{attribute 'linkalways'} 
{attribute 'no_explicit_call' := 'This FB is a CLASS and must be accessed using methods or properties'}
{attribute 'enable_dynamic_creation'}
FUNCTION_BLOCK _WORD EXTENDS NumericDatatypeBase
VAR
	localData : WORD;
	activeData : REFERENCE TO WORD REF= localData;
END_VAR

PROPERTY PUBLIC Address : PVOID
GET
Address := ADR(activeData);
END_GET
END_PROPERTY

METHOD PUBLIC ClearReference
VAR_INPUT
END_VAR
activeData REF= localData;
END_METHOD

METHOD PUBLIC Clone : I_Datatype
VAR
    pClone : POINTER TO _WORD;
END_VAR
pClone := __NEW(_WORD(InitialValue := Value));
Clone := pClone^;
END_METHOD

METHOD FB_init : BOOL
VAR_INPUT
	bInitRetains : BOOL; // if TRUE, the retain variables are initialized (warm start / cold start)
	bInCopyCode : BOOL;  // if TRUE, the instance afterwards gets moved WORDo the copy code (online change)
	InitialValue : WORD;
END_VAR
localData := InitialValue;
END_METHOD

PROPERTY PUBLIC IsEven : BOOL
GET
IsEven := (Value mod 2) = 0;
END_GET
END_PROPERTY

PROPERTY PUBLIC IsFloat : BOOL
GET
IsFloat := FALSE;
END_GET
END_PROPERTY

PROPERTY PUBLIC IsSigned : BOOL
GET
IsSigned := FALSE;
END_GET
END_PROPERTY

METHOD PUBLIC MakeReferenceTo
VAR_INPUT
	ReferenceTarget : REFERENCE TO WORD;
END_VAR
activeData REF= ReferenceTarget;
END_METHOD

PROPERTY PUBLIC MaxValue : WORD
GET
MaxValue :=  DatatypeLimits.WORD_MAX_VALUE;
END_GET
END_PROPERTY

PROPERTY PUBLIC MinValue : WORD
GET
MinValue := DatatypeLimits.WORD_MIN_VALUE;
END_GET
END_PROPERTY

METHOD PROTECTED SerializeMaxValue
VAR_INPUT
	Serializer : I_Serializer;
END_VAR
Serializer.AddWord(MaxValue);
END_METHOD

METHOD PROTECTED SerializeMinValue
VAR_INPUT
	Serializer : I_Serializer;
END_VAR
Serializer.AddWord(MinValue);
END_METHOD

METHOD PUBLIC SerializeWith
VAR_INPUT
	Serializer : I_Serializer;
END_VAR
Serializer.AddWord(activeData);
END_METHOD

PROPERTY PUBLIC Size : UDINT
GET
Size := SIZEOF(activeData);
END_GET
END_PROPERTY

METHOD TryDeserializeFrom : BOOL
VAR_INPUT
	Deserializer : I_Deserializer;
	Feedback : I_DeserializerFeedback;
END_VAR
TryDeserializeFrom := Deserializer.TryGetWord(activeData, Feedback);
END_METHOD

METHOD TryMakeReferenceTo : BOOL
VAR_INPUT
	Target : I_Datatype;
END_VAR
VAR
	pTargetData : POINTER TO WORD;
END_VAR
IF NOT IsEquivalentTo(Target) THEN
	RETURN;
END_IF

pTargetData := Target.Address;
activeData REF= pTargetData^;
TryMakeReferenceTo := TRUE;
END_METHOD

PROPERTY PUBLIC TypeName : T_MAXSTRING
GET
TypeName := 'WORD';
END_GET
END_PROPERTY

PROPERTY PUBLIC Value : REFERENCE TO WORD
GET
Value REF= activeData;
END_GET
END_PROPERTY

END_FUNCTION_BLOCK

(* stored: Version 1.1.0.1, ProductVersion 3.1.4024.13
   POU _WORD: Id {785b4543-75b4-4d22-ba61-129866dbb78f}, SpecialFunc None
   Folder Constructor: Id {2bc942c9-15ef-443c-86a0-0ba3d6f8acbf}
   Folder Protected: Id {a63c5a23-6486-48b9-8570-ceb36a757b18}
   Property Address: Id {dde93b64-d15e-4c83-a1c7-9a71a5203dbd}
   Get Get: Id {15831d15-e22a-4e2b-bf87-eb7a5f0007f2}
   Method ClearReference: Id {006bc84c-7a71-4a67-9fcd-5c4ef11d0d04}
   Method Clone: Id {3ad80d2a-a76e-4b25-a839-a3445f1727ce}
   Method FB_init: Id {25cb8094-357a-4e3b-b5fe-15624aba575c}
   Property IsEven: Id {9e740dfe-6f0d-0e02-2109-625bfe544a0f}
   Get Get: Id {9d1a7e75-20cb-0222-3716-8a44a1b6f195}
   Property IsFloat: Id {9031cfa6-6438-4d3a-94a7-7b1d37055da1}
   Get Get: Id {7390886d-ad43-4baa-ba6b-c5b294a25c3a}
   Property IsSigned: Id {75ebcade-d7b4-4897-8091-d07bca5214dc}
   Get Get: Id {4bd4aebb-55aa-4478-8ca6-2f0f9370ffc2}
   Method MakeReferenceTo: Id {4c888c95-4902-445b-bffe-15128e43a6d3}
   Property MaxValue: Id {df183709-e5a2-44ff-87d7-9368105dab63}
   Get Get: Id {28fd4b6d-ce35-4c59-a813-06cb5556e621}
   Property MinValue: Id {37d80b64-8e58-4f9d-9f8a-37a1acd57600}
   Get Get: Id {788b7e61-0ffc-4237-a55d-41150ae7f999}
   Method SerializeMaxValue: Id {6cf67daa-fa5f-4f6b-b5c0-6a8a33d5e532}
   Method SerializeMinValue: Id {9e6ebab6-c168-44a3-9857-d853802e8cef}
   Method SerializeWith: Id {ff03b8e8-977c-4201-aaa1-7b0e153d93cd}
   Property Size: Id {2bdd1b22-de81-4397-8b38-532f4fd909a3}
   Get Get: Id {b95c9a04-8956-463c-ac0e-bd89d4a7164f}
   Method TryDeserializeFrom: Id {00f03103-9e65-4c26-99af-92a5fda659ca}
   Method TryMakeReferenceTo: Id {a85aab6e-0868-49b5-a56c-8d1f3422f73f}
   Property TypeName: Id {ea67172d-3b40-4ad0-ae37-3ab08a0b7855}
   Get Get: Id {b997ca83-025a-40c6-96c4-34086c410ab4}
   Property Value: Id {e62bcf86-3880-4080-9eae-bbad242889c9}
   Get Get: Id {466faa1b-1333-47fa-aaf0-4b401c13734f} *)
